// TIA Portal V18 export
// export: Created 2026-06-22T15:41:34.9359236Z, ExportSetting WithDefaults, DisplayName Totally Integrated Automation Portal, DisplayVersion V18, DisplayName TIA Portal Openness, DisplayVersion V18, DisplayName TIA Portal Version Control Interface, DisplayVersion V18, DisplayName STEP 7 Professional, DisplayVersion V18, DisplayName STEP 7 Safety, DisplayVersion V18, DisplayName WinCC Professional, DisplayVersion V18
VAR_GLOBAL   // PLC tag table "Encoder_Tags"
   HSC_1_Value AT %ID1000 : DInt;   // Giá trị đếm xung thời kỳ thực từ bộ đếm tốc độ cao HSC1   {ExternalWritable false}
END_VAR
